(* IEC 61131-3 sources: Modular-Warehouse-Automation-Architecture/plc_code, 3 files *)

(* ---- FB_AlarmManager.st ---- *)
FUNCTION_BLOCK FB_AlarmManager
VAR_INPUT
    FaultInput : BOOL;
END_VAR

VAR_OUTPUT
    AlarmActive : BOOL;
    AlarmCode   : INT;
END_VAR

IF FaultInput THEN
    AlarmActive := TRUE;
    AlarmCode := 1001; // Example fault code
ELSE
    AlarmActive := FALSE;
    AlarmCode := 0;
END_IF;

(* ---- FB_ConveyorControl.st ---- *)
FUNCTION_BLOCK FB_ConveyorControl
VAR_INPUT
    StartCmd   : BOOL;
    StopCmd    : BOOL;
    FaultReset : BOOL;
END_VAR

VAR_OUTPUT
    ConveyorRun : BOOL;
    FaultActive : BOOL;
END_VAR

VAR
    InternalFault : BOOL;
END_VAR

IF FaultReset THEN
    InternalFault := FALSE;
END_IF;

IF StartCmd AND NOT StopCmd AND NOT InternalFault THEN
    ConveyorRun := TRUE;
ELSIF StopCmd THEN
    ConveyorRun := FALSE;
END_IF;

// Simulated fault condition placeholder
IF ConveyorRun = TRUE AND FALSE THEN
    InternalFault := TRUE;
END_IF;

FaultActive := InternalFault;

(* ---- FB_StateMachine.st ---- *)
FUNCTION_BLOCK FB_StateMachine
VAR_INPUT
    Start : BOOL;
    Stop  : BOOL;
END_VAR

VAR_OUTPUT
    State : INT;
END_VAR

// States: 0=Idle, 1=Running, 2=Stopped
IF Start THEN
    State := 1;
END_IF;

IF Stop THEN
    State := 2;
END_IF;

IF NOT Start AND NOT Stop THEN
    State := 0;
END_IF;
